INTERFACE I_Indicator

METHOD Flash
VAR_INPUT
END_VAR
END_METHOD

METHOD TurnOff
VAR_INPUT
END_VAR
END_METHOD

METHOD TurnOn
VAR_INPUT
END_VAR
END_METHOD

END_INTERFACE

(* stored: Version 1.1.0.1
   Itf I_Indicator: Id {ccfdfa01-d0e3-4f35-b29d-a16def021e32}
   Method Flash: Id {9b233834-00bb-4ee5-bdce-784659a71445}
   Method TurnOff: Id {e910b58a-e84f-4acf-8628-412e3b28658a}
   Method TurnOn: Id {6b06190f-522d-4c7a-87b4-da85a0178d06} *)
